{attribute 'qualified_only'}
{attribute 'strict'}
TYPE TopLevelSTM :
(
	STARTUP,
	READY,
	OPERATIONAL,
	SHUTDOWN,
	ERROR
)USINT;
END_TYPE

(* stored: Version 1.1.0.1, ProductVersion 3.1.4024.12
   DUT TopLevelSTM: Id {ae2f80c0-7219-4e14-b5e1-3d29d14ade86} *)
